{attribute 'linkalways'} 
{attribute 'no_explicit_call' := 'This FB is a CLASS and must be accessed using methods or properties'}
{attribute 'enable_dynamic_creation'}
FUNCTION_BLOCK Node_F_VN_SetAt_TcVnVector2_REAL EXTENDS VisionNode
VAR
    aElement : _TcVnVector2_REAL;
    ipContainer : _ITcVnContainer;
    nIndex : _ULINT(0);
    hrPrev : _HRESULT(S_OK);
    hresult : _HRESULT(S_OK);
END_VAR

METHOD PUBLIC  Clone : I_Node
VAR
	pNode : POINTER TO Node_F_VN_SetAt_TcVnVector2_REAL;
END_VAR
pNode := __NEW(Node_F_VN_SetAt_TcVnVector2_REAL);
Clone := pNode^;
END_METHOD

METHOD FB_init : BOOL
VAR_INPUT
	bInitRetains : BOOL; // if TRUE, the retain variables are initialized (warm start / cold start)
	bInCopyCode : BOOL;  // if TRUE, the instance afterwards gets moved into the copy code (online change)
END_VAR
AddInput('aElement', aElement);
AddInput('ipContainer', ipContainer);
AddInput('nIndex', nIndex);
AddInput('hrPrev', hrPrev);
AddOutput('ipContainer', ipContainer);
AddOutput('hresult',hresult);
END_METHOD

METHOD PROTECTED OnExecute : HRESULT
hresult.Value := F_VN_SetAt_TcVnVector2_REAL(
    aElement := aElement.Value,
    ipContainer := ipContainer.Value,
    nIndex := nIndex.Value,
    hrPrev:= hrPrev.Value);
END_METHOD

METHOD PUBLIC PreExecutionCheck
VAR_INPUT
	Check : I_PreExecutionChecks;
END_VAR
Check.IsTrue(ipContainer.IsValid, 'ipContainer must be a valid container');
END_METHOD

END_FUNCTION_BLOCK

(* stored: Version 1.1.0.1, ProductVersion 3.1.4024.13
   POU Node_F_VN_SetAt_TcVnVector2_REAL: Id {f399fa5f-01e4-46e1-bb52-7827f524108b}, SpecialFunc None
   Folder Constructor: Id {88ee8e6a-11e9-4540-bc35-d67f20642217}
   Method Clone: Id {77b44394-fd85-4b5e-8ba7-629d76735551}
   Method FB_init: Id {0e0ae33c-d2d6-4ed0-81b3-807d235f67df}
   Method OnExecute: Id {7087f032-c190-4be0-8bca-323ac92bef2e}
   Method PreExecutionCheck: Id {eee8f7ac-ca39-41b1-ae24-7016e5c55347} *)
